(* PLC project v0.6.04_CycleSemiAuto.project, CODESYS CODESYS V3.5 SP19 Patch 1 *)
(* stored: creationDateTime 2026-08-14T20:21:08.548739, modificationDateTime 2026-08-14T20:21:08.548739 *)

(* ═══════════════════════════════════════════════════════════════ 🧪 FB_Sim_Translation — Progression capteurs simulés M3 ─────────────────────────────────────────────────────────────── 🎯 Rôle : Produit les cinq capteurs de position M3 par progression continue de Trémie vers Maintenance. Le modèle ne publie que les six mots valides de FB_Translation_PositionDecoder : 11111 → 01111 → 00111 → 00011 → 00001 → 00000. 🔒 Le modèle est une source d'entrée confinée derrière HwIn ; il ne pilote aucune sortie réelle. Un override manuel valide est appliqué par FB_SimBench, pas par ce FB. 📄 Docs : DOC/AF/AF_Partie-13_Fonction_Simulation_v2.3.md DOC/AF/AF_Partie-11_Fonction_Translation_v2.2.md ═══════════════════════════════════════════════════════════════ *)
FUNCTION_BLOCK FB_Sim_Translation
  VAR_INPUT
    Enable : BOOL;  (* TRUE = modèle actif *)
    Direction : INT;  (* +1 = vers Trémie ; -1 = vers Maintenance ; 0 = maintien position *)
    SpeedRefPct : REAL;  (* Magnitude commande 0..100 %, bornée avant calcul *)
    FullTravelTimeS : REAL := 8;  (* Temps complet Trémie→Maintenance à 100 %, simulation seulement *)
  END_VAR
  VAR_OUTPUT
    PosTremie : BOOL;  (* Bit4 du mot capteurs *)
    PosPV : BOOL;  (* Bit3 du mot capteurs *)
    PosP2 : BOOL;  (* Bit2 du mot capteurs (point matériel PVP2) *)
    PosP1 : BOOL;  (* Bit1 du mot capteurs *)
    PosMaintenance : BOOL;  (* Bit0 du mot capteurs *)
  END_VAR
  VAR
    instCycleTime : FB_CycleTime;
    PositionProgress : REAL;  (* 0=Trémie ... 5=Maintenance *)
    SpeedPctBounded : REAL;
    PositionIncrement : REAL;
    Initialized : BOOL := FALSE;
    CST_PositionAtTremie : REAL := 0;
    CST_PositionAtPV : REAL := 1;
    CST_PositionAtP2 : REAL := 2;
    CST_PositionAtP1 : REAL := 3;
    CST_PositionAtMaintenance : REAL := 5;
    CST_PositionSegmentCount : REAL := 5;
    CST_MinFullTravelTimeS : REAL := 0.1;  (* Protection division : modèle sans dynamique sous ce seuil *)
  END_VAR

            

// === IMPLEMENTATION ===

IF NOT Enable THEN
    // Prochain démarrage déterministe sur P2, comme l'ancien modèle de banc.
    PositionProgress := CST_PositionAtP2;
    Initialized := FALSE;
    PosTremie := FALSE;
    PosPV := FALSE;
    PosP2 := FALSE;
    PosP1 := FALSE;
    PosMaintenance := FALSE;
    RETURN;
END_IF;

IF NOT Initialized THEN
    PositionProgress := CST_PositionAtP2;
    Initialized := TRUE;
END_IF;

instCycleTime(DefaultValueS := 0.010);
SpeedPctBounded := LIMIT(0.0, ABS(SpeedRefPct), 100.0);

// Une vitesse à 100 % parcourt les cinq segments uniformes pendant FullTravelTimeS.
// Direction sémantique : +1 réduit la progression vers Trémie ; -1 l'augmente vers Maintenance.
IF FullTravelTimeS >= CST_MinFullTravelTimeS THEN
    PositionIncrement := (SpeedPctBounded / 100.0)
                         * (CST_PositionSegmentCount / FullTravelTimeS)
                         * instCycleTime.CycleTimeS;
ELSE
    PositionIncrement := 0.0;
END_IF;

IF Direction = 1 THEN
    PositionProgress := MAX(CST_PositionAtTremie, PositionProgress - PositionIncrement);
ELSIF Direction = -1 THEN
    PositionProgress := MIN(CST_PositionAtMaintenance, PositionProgress + PositionIncrement);
END_IF;

// Réinitialisation explicite : aucune valeur transitoire héritée d'une zone précédente.
PosTremie := FALSE;
PosPV := FALSE;
PosP2 := FALSE;
PosP1 := FALSE;
PosMaintenance := FALSE;

// Chaque intervalle correspond à un seul mot thermomètre valide.
IF PositionProgress <= CST_PositionAtTremie THEN
    PosTremie := TRUE;
    PosPV := TRUE;
    PosP2 := TRUE;
    PosP1 := TRUE;
    PosMaintenance := TRUE;
ELSIF PositionProgress <= CST_PositionAtPV THEN
    PosPV := TRUE;
    PosP2 := TRUE;
    PosP1 := TRUE;
    PosMaintenance := TRUE;
ELSIF PositionProgress <= CST_PositionAtP2 THEN
    PosP2 := TRUE;
    PosP1 := TRUE;
    PosMaintenance := TRUE;
ELSIF PositionProgress <= CST_PositionAtP1 THEN
    PosP1 := TRUE;
    PosMaintenance := TRUE;
ELSIF PositionProgress < CST_PositionAtMaintenance THEN
    PosMaintenance := TRUE;
END_IF;

          
END_FUNCTION_BLOCK

(* ═══════════════════════════════════════════════════════════════ ⏱️ FB_CycleTime — Mesure du temps de cycle réel de la tâche ─────────────────────────────────────────────────────────────── 📄 Doc métier : DOC/AF/AF_Partie-08_Fonction_Joystick_v2.0.md §2 (base de temps utilisée par FB_Filter_PT1, composé dans FB_Joystick) ═══════════════════════════════════════════════════════════════ *)
FUNCTION_BLOCK FB_CycleTime
  VAR_INPUT
    DefaultValueS : REAL := 0.004;  (* Valeur de secours par défaut (ex. 4ms) *)
  END_VAR
  VAR_OUTPUT
    CycleTimeS : REAL;  (* Temps écoulé réel calculé (secondes) *)
  END_VAR
  VAR
    TimeCurrent : TIME;  (* Temps système actuel *)
    TimeLast : TIME;  (* Empreinte de temps du cycle précédent *)
    DeltaTimeMs : UDINT;  (* Écart brut calculé (ms) *)
    InitDone : BOOL;  (* Drapeau d'initialisation du premier cycle *)
  END_VAR

            

// 1. ACQUISITION DU TEMPS SYSTÈME
TimeCurrent := TIME();

// 2. INITIALISATION UNIQUE AU PREMIER CYCLE
IF NOT InitDone THEN
    TimeLast := TimeCurrent;
    InitDone := TRUE;
    CycleTimeS := DefaultValueS;
    RETURN;
END_IF;

// 3. CALCUL DU DELTA EN MILLISECONDES
DeltaTimeMs := TIME_TO_UDINT(TimeCurrent - TimeLast);

// 4. CONVERSION ET CHARGE DE SECOURS
IF DeltaTimeMs > 0 THEN
    CycleTimeS := UDINT_TO_REAL(DeltaTimeMs) / 1000.0;
ELSE
    CycleTimeS := DefaultValueS;
END_IF;

// 5. ARCHIVAGE POUR LE PROCHAIN CYCLE
TimeLast := TimeCurrent;

          
END_FUNCTION_BLOCK
